// Core §3.15.1a — CM base for ASCII request/response devices over I_ByteChannel
// (vision sensors, code readers, gauges). One-outstanding-request state machine:
// SendRequest -> await terminated response -> _M_OnResponse hook; silence -> fault
// 10402. The framing and request rules are FB_AsciiLink's, shared with connectors
// (§1.1 O9); this CM adds what a CM owns: its faults and its bounded reconnect.
// Written ONCE against the neutral seam: porting = swap the channel (O4/O8).
FUNCTION_BLOCK ABSTRACT FB_AsciiDeviceCM EXTENDS FB_ControlModuleBase
VAR
    Host        : STRING(80);          // §3.8 config (per deployment)
    Port        : UINT;
    Terminator  : STRING(2) := '$R';   // CR default; device profile may override
    RespTimeout : TIME := T#2S;
    LinkState   : E_ByteChannelState;  // published (Annex D link facet)
    LastResponse: STRING(255);         // published (diagnosis)
END_VAR
VAR
    {attribute 'OPC.UA.DA' := '0'}
    _link      : FB_AsciiLink;
    _tRetry    : TON;
    _retryMs   : TIME := T#500MS;       // bounded backoff (doubles to 10s)
    _openTried : BOOL;                  // backoff spaces RE-tries; the first Open is immediate
END_VAR

;  // driven via Cyclic (base) -> OnCyclic below

// wire the transport + endpoint. Call from the profile's Setup after _M_SetName.
METHOD SetupDevice : BOOL
VAR_INPUT
    Chan : I_ByteChannel;
    DevHost : STRING(80);
    DevPort : UINT;
END_VAR
IF Chan = 0 OR DevHost = '' THEN
    _M_FaultN(PL_TcpDevReasons.DEV_CFG_INVALID, 'std.error.deviceConnectionNotConfigured');
    SetupDevice := FALSE;
    RETURN;
END_IF
_link.M_Bind(Chan := Chan);
Host := DevHost;
Port := DevPort;
SetupDevice := TRUE;
END_METHOD

// channel management + RX framing. Profiles override _M_OnResponse, not this.
METHOD PROTECTED OnCyclic : DINT
VAR
    evt : E_AsciiLinkEvent;
END_VAR
OnCyclic := SUPER^.OnCyclic();
_link.Terminator := Terminator;
_link.RespTimeout := RespTimeout;
evt := _link.M_Tick();
LinkState := _link.State;
IF LinkState = E_ByteChannelState.CLOSED THEN
    IF NOT _openTried THEN
        _openTried := TRUE;                        // first sight of CLOSED: connect NOW
        _link.M_Open(Host := Host, Port := Port);
        LinkState := _link.State;                  // a synchronous transport is OPEN this scan
    ELSE
        _tRetry(IN := TRUE, PT := _retryMs);       // failed before: bounded backoff (§3.15.2 spirit)
        IF _tRetry.Q THEN
            _tRetry(IN := FALSE);
            _link.M_Open(Host := Host, Port := Port);
            LinkState := _link.State;
            IF _retryMs < T#10S THEN
                _retryMs := _retryMs * 2;
            END_IF
        END_IF
    END_IF
ELSIF LinkState = E_ByteChannelState.OPEN THEN
    _openTried := FALSE;
    _retryMs := T#500MS;
END_IF
CASE evt OF
    E_AsciiLinkEvent.NONE:
        ;
    E_AsciiLinkEvent.RESPONSE:
        LastResponse := _link.LastResponse;
        _M_OnResponse(Response := _link.Response);
    E_AsciiLinkEvent.OVERFLOW:
        _M_FaultN(PL_TcpDevReasons.DEV_RX_OVERFLOW, 'std.error.deviceResponseOverflow');
    E_AsciiLinkEvent.CHANNEL_FAULT:
        _M_FaultN(PL_TcpDevReasons.DEV_CHANNEL_FAULT, 'std.error.transportChannelFault');
    E_AsciiLinkEvent.TIMEOUT:
        _M_FaultN(PL_TcpDevReasons.DEV_RESP_TIMEOUT, 'std.error.deviceResponseTimeout');
ELSE
    _M_FaultN(PL_TcpDevReasons.DEV_CHANNEL_FAULT, 'std.error.byteChannelStateInvalid');
END_CASE
END_METHOD

// issue one request (terminator appended). FALSE if not connected or one pending.
METHOD SendRequest : BOOL
VAR_INPUT
    Text : STRING(250);
END_VAR
IF NOT _link.M_IsOpen() THEN
    _M_FaultN(PL_TcpDevReasons.DEV_NOT_CONNECTED, 'std.error.deviceNotConnected');
    SendRequest := FALSE;
    RETURN;
END_IF
// A pending request is the one-outstanding contract, not a fault: refused quietly.
_link.Terminator := Terminator;
SendRequest := _link.M_Send(Text := Text);
END_METHOD

// profile hook: parse one terminated response. Raise DEV_PROTOCOL on garbage.
METHOD PROTECTED _M_OnResponse
VAR_INPUT
    Response : STRING(255);
END_VAR
;
END_METHOD

END_FUNCTION_BLOCK

(* stored: Version 1.1.0.1, ProductVersion 3.1.4024.12
   POU FB_AsciiDeviceCM: Id {fbdfe34e-2b13-471d-9c7e-f6c09e1b07f2}, SpecialFunc None
   Method SetupDevice: Id {2ab03770-7cce-43e3-a8b7-260bc7ab0b22}
   Method OnCyclic: Id {641940cd-41bc-490f-a5b9-7fd36e427088}
   Method SendRequest: Id {762283fc-05d7-4631-9d26-11346d11feba}
   Method _M_OnResponse: Id {458bd92a-0a1d-42f4-9a5c-8b7706bcaf76} *)
